% RSLogix 500 project UNTITLED_BAK000.RSS, saved by version 8.30.00.16 %
PROJECT "UNTITLED"    % processor: Bul.1763 MicroLogix 1100 Series B %

PROGRAM FILES
  LAD 2   18 rungs

DATA FILES
  O0 OUTPUT  4 elements
  I1 INPUT  6 elements
  S2 STATUS  66 elements
  B3 BINARY  20 elements
  T4 TIMER  1 elements
  C5 COUNTER  1 elements
  R6 CONTROL  1 elements
  N7 INTEGER  1 elements
  F8 FLOAT  1 elements

LADDER 2
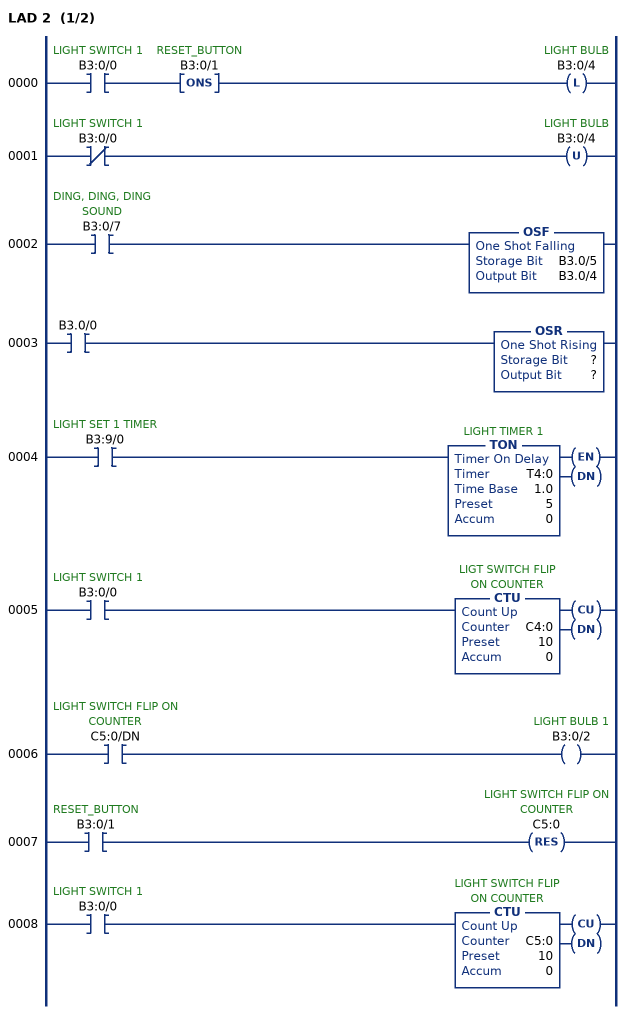
% Rung: 0 %  % edit flag set %
SOR XIC B3:0/0 ONS B3:0/1 OTL B3:0/4 EOR
%   B3:0/0  "LIGHT SWITCH 1" %
%   B3:0/1  RESET_BUTTON %
%   B3:0/4  "LIGHT BULB" %
% Rung: 1 %  % edit flag set %
SOR XIO B3:0/0 OTU B3:0/4 EOR
%   B3:0/0  "LIGHT SWITCH 1" %
%   B3:0/4  "LIGHT BULB" %
% Rung: 2 %  % edit flag set %
SOR XIC B3:0/7 OSF B3.0/5 B3.0/4 EOR
%   B3:0/7  "DING, DING, DING SOUND" %
% Rung: 3 %  % edit flag set %
SOR XIC B3.0/0 OSR ? ? EOR
% Rung: 4 %  % edit flag set %
SOR XIC B3:9/0 TON T4:0 1.0 5 0 EOR
%   B3:9/0  "LIGHT SET 1 TIMER" %
%   T4:0  "LIGHT TIMER 1" %
% Rung: 5 %  % edit flag set %
SOR XIC B3:0/0 CTU C4:0 10 0 EOR
%   B3:0/0  "LIGHT SWITCH 1" %
%   C4:0  "LIGT SWITCH FLIP ON COUNTER" %
% Rung: 6 %  % edit flag set %
SOR XIC C5:0/DN OTE B3:0/2 EOR
%   C5:0  "LIGHT SWITCH FLIP ON COUNTER" %
%   B3:0/2  "LIGHT BULB 1" %
% Rung: 7 %  % edit flag set %
SOR XIC B3:0/1 RES C5:0 EOR
%   B3:0/1  RESET_BUTTON %
%   C5:0  "LIGHT SWITCH FLIP ON COUNTER" %
% Rung: 8 %  % edit flag set %
SOR XIC B3:0/0 CTU C5:0 10 0 EOR
%   B3:0/0  "LIGHT SWITCH 1" %
%   C5:0  "LIGHT SWITCH FLIP ON COUNTER" %

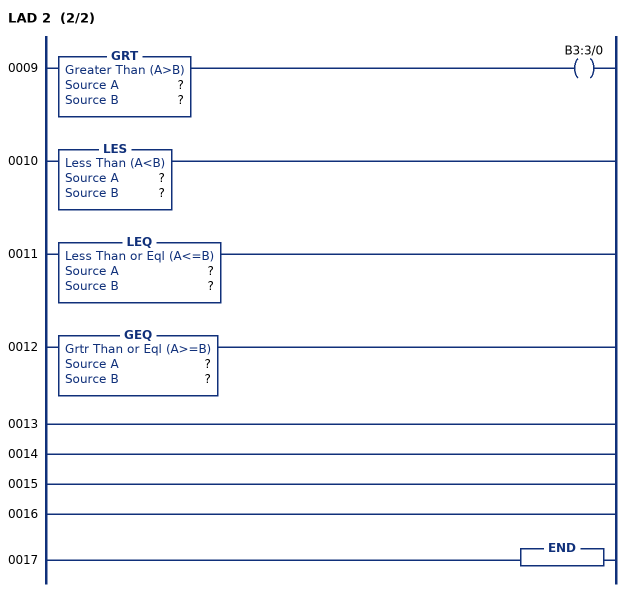
% Rung: 9 %  % edit flag set %
SOR GRT ? ? OTE B3:3/0 EOR
% Rung: 10 %  % edit flag set %
SOR LES ? ? EOR
% Rung: 11 %  % edit flag set %
SOR LEQ ? ? EOR
% Rung: 12 %  % edit flag set %
SOR GEQ ? ? EOR
% Rung: 13 %  % edit flag set %
SOR EOR
% Rung: 14 %  % edit flag set %
SOR EOR
% Rung: 15 %  % edit flag set %
SOR EOR
% Rung: 16 %  % edit flag set %
SOR EOR
% Rung: 17 %
SOR END EOR

OTHER DOCUMENTED ADDRESSES
  B3:3/2  "LIGT BULB 1-1"
